PROGRAM PRG_Events
VAR
    aWarningEvents : ARRAY[0..4, 0..100] OF BOOL;
// 	sHeaterMinimum : STRING(32);
// 	sHeaterCurrent : STRING(32);
    fbEventsManager : FB_EventsManager;
    tonUpSupplyLost : TON;
    tonUsSupplyLost : TON;
    ton48VSupplyLost : TON;
    tonIndexPositionInvalid : TON;

    // Short-lived operator feedback for Heat Stake settings transactions.
    tpHeatStakeSettingsSaved : TP;
    tpHeatStakeSettingsRejected : TP;
    tpHeatStakeSettingsSaveFailed : TP;
END_VAR

GVL_MASTER.stStationEvents[0].aEvents[0].bFault := TRUE;
GVL_MASTER.stStationEvents[0].aEvents[0].bEventFlag :=
    (NOT GVL_MASTER.stInputs.bEmergencyStopChannel1 OR NOT GVL_MASTER.stInputs.bEmergencyStopChannel2)
    AND NOT GVL_MASTER.stInputs.stSafety.bSafetyOk;
GVL_MASTER.stStationEvents[0].aEvents[0].bEventText := 'E-stop activated';
GVL_MASTER.stStationEvents[0].aEvents[0].sSolution := 'Release E-stop and reset Safety';

GVL_MASTER.stStationEvents[0].aEvents[1].bFault := TRUE;
GVL_MASTER.stStationEvents[0].aEvents[1].bEventFlag :=
    (NOT GVL_MASTER.stInputs.bMainDoorChannel1 OR NOT GVL_MASTER.stInputs.bMainDoorChannel2)
    AND NOT GVL_MASTER.stInputs.stSafety.bSafetyOk;
GVL_MASTER.stStationEvents[0].aEvents[1].bEventText := 'Main door safety circuit open';
GVL_MASTER.stStationEvents[0].aEvents[1].sSolution := 'Close main door and reset Safety';


GVL_MASTER.stStationEvents[0].aEvents[2].bFault := TRUE;
GVL_MASTER.stStationEvents[0].aEvents[2].bEventFlag :=
    (NOT GVL_MASTER.stInputs.bLeftFlapChannel1 OR NOT GVL_MASTER.stInputs.bLeftFlapChannel2)
    AND NOT GVL_MASTER.stInputs.stSafety.bSafetyOk
    AND (GVL_MASTER.stStatus.eMachineState <> E_MachineState.PowerUp);
GVL_MASTER.stStationEvents[0].aEvents[2].bEventText := 'Right safety flap active';
GVL_MASTER.stStationEvents[0].aEvents[2].sSolution := 'Clear right flap and reset Safety';


GVL_MASTER.stStationEvents[0].aEvents[3].bFault := TRUE;
GVL_MASTER.stStationEvents[0].aEvents[3].bEventFlag :=
    (NOT GVL_MASTER.stInputs.bRightFlapChannel1 OR NOT GVL_MASTER.stInputs.bRightFlapChannel2)
    AND NOT GVL_MASTER.stInputs.stSafety.bSafetyOk
    AND (GVL_MASTER.stStatus.eMachineState <> E_MachineState.PowerUp);
GVL_MASTER.stStationEvents[0].aEvents[3].bEventText := 'Left safety flap active';
GVL_MASTER.stStationEvents[0].aEvents[3].sSolution := 'Clear left flap and reset Safety';


GVL_MASTER.stStationEvents[0].aEvents[4].bCycleStopRequest := TRUE;
GVL_MASTER.stStationEvents[0].aEvents[4].bEventFlag := GVL_MASTER.stCommand.bStop;
GVL_MASTER.stStationEvents[0].aEvents[4].bEventText := 'Cycle stop requested';
GVL_MASTER.stStationEvents[0].aEvents[4].sSolution := 'Wait for cycle to stop';

GVL_MASTER.stStationEvents[0].aEvents[5].bFault := TRUE;
GVL_MASTER.stStationEvents[0].aEvents[5].bEventFlag := GVL_MASTER.stStatus.bInitialisationTimeoutFault;
GVL_MASTER.stStationEvents[0].aEvents[5].bEventText := 'System initialisation timeout';
GVL_MASTER.stStationEvents[0].aEvents[5].sSolution := 'Check initialisation conditions';


GVL_MASTER.stStationEvents[0].aEvents[6].bFault := TRUE;
GVL_MASTER.stStationEvents[0].aEvents[6].bEventFlag := GVL_MASTER.stStatus.bStoppingTimeoutFault;
GVL_MASTER.stStationEvents[0].aEvents[6].bEventText := 'System stopping timeout';
GVL_MASTER.stStationEvents[0].aEvents[6].sSolution := 'Check index and machine safe state';


// Main-door supervision already causes immediate Fault; expose its actual cause.
GVL_MASTER.stStationEvents[0].aEvents[22].bFault := TRUE;
GVL_MASTER.stStationEvents[0].aEvents[22].bCycleStopRequest := FALSE;
GVL_MASTER.stStationEvents[0].aEvents[22].bEventFlag := GVL_MASTER.stStatus.stMainDoorLock.bFaulted;
GVL_MASTER.stStationEvents[0].aEvents[22].bEventText := CONCAT('Main door: ', GVL_MASTER.stStatus.stMainDoorLock.sMessage);
GVL_MASTER.stStationEvents[0].aEvents[22].sSolution := 'Check door/lock feedback and requested lock state; correct cause before Reset.';

tonUpSupplyLost(IN := NOT GVL_MASTER.stInputs.bUp24VPowerSupplyOk AND (GVL_MASTER.stStatus.eMachineState <> E_MachineState.PowerUp), PT := T#1S);

GVL_MASTER.stStationEvents[0].aEvents[7].bFault := TRUE;
GVL_MASTER.stStationEvents[0].aEvents[7].bEventFlag := tonUpSupplyLost.Q;
GVL_MASTER.stStationEvents[0].aEvents[7].bEventText := '24 V Up supply fault';
GVL_MASTER.stStationEvents[0].aEvents[7].sSolution := 'Check 24 V Up power supply';


tonUsSupplyLost(IN := NOT GVL_MASTER.stInputs.bUs24VPowerSupplyOk AND (GVL_MASTER.stStatus.eMachineState <> E_MachineState.PowerUp), PT := T#1S);

GVL_MASTER.stStationEvents[0].aEvents[8].bFault := TRUE;
GVL_MASTER.stStationEvents[0].aEvents[8].bEventFlag := tonUsSupplyLost.Q;
GVL_MASTER.stStationEvents[0].aEvents[8].bEventText := '24 V Us supply fault';
GVL_MASTER.stStationEvents[0].aEvents[8].sSolution := 'Check 24 V Us power supply';


ton48VSupplyLost(IN := NOT GVL_MASTER.stInputs.b48VPowerSupplyOk AND (GVL_MASTER.stStatus.eMachineState <> E_MachineState.PowerUp), PT := T#1S);

GVL_MASTER.stStationEvents[0].aEvents[9].bFault := TRUE;
GVL_MASTER.stStationEvents[0].aEvents[9].bEventFlag := ton48VSupplyLost.Q;
GVL_MASTER.stStationEvents[0].aEvents[9].bEventText := '48 V Up supply fault';
GVL_MASTER.stStationEvents[0].aEvents[9].sSolution := 'Check 48 V power supply';


tonIndexPositionInvalid(IN := GVL_MASTER.stInputs.bIndexReady AND GVL_MASTER.stInputs.bIndexLocked AND (GVL_MASTER.stInputs.eIndexPosition = E_TablePosition.Unknown), PT := T#500MS);

GVL_MASTER.stStationEvents[2].aEvents[0].bFault := TRUE;
GVL_MASTER.stStationEvents[2].aEvents[0].bEventFlag := tonIndexPositionInvalid.Q;
GVL_MASTER.stStationEvents[2].aEvents[0].bEventText := 'Index position sensors invalid';
GVL_MASTER.stStationEvents[2].aEvents[0].sSolution := 'Check index position sensors';



// -----------------------------------------------------------------------------
// PATCH PRESS STATION SUPPORT CYLINDERS
// Station group [3] is reserved here for process-station pneumatic faults.
// Each event is a machine fault and therefore participates in the existing
// bEventFault -> bSafetyDropRequest -> Immediate Fault chain.
// -----------------------------------------------------------------------------

// Patch Dispense support cylinder.
GVL_MASTER.stStationEvents[3].aEvents[0].bFault := TRUE;
GVL_MASTER.stStationEvents[3].aEvents[0].bEventFlag :=
    GVL_MASTER.stStatus.stPatchDispense.eSupportFault = E_SupportCylinderFault.ExtendTimeout;
GVL_MASTER.stStationEvents[3].aEvents[0].bEventText := 'Patch Dispense support cylinder UP feedback timeout';
GVL_MASTER.stStationEvents[3].aEvents[0].sSolution := 'Check UP sensor, air pressure, tubing, valve and cylinder mechanics';

GVL_MASTER.stStationEvents[3].aEvents[1].bFault := TRUE;
GVL_MASTER.stStationEvents[3].aEvents[1].bEventFlag :=
    GVL_MASTER.stStatus.stPatchDispense.eSupportFault = E_SupportCylinderFault.RetractTimeout;
GVL_MASTER.stStationEvents[3].aEvents[1].bEventText := 'Patch Dispense support cylinder DOWN feedback timeout';
GVL_MASTER.stStationEvents[3].aEvents[1].sSolution := 'Check DOWN sensor, air pressure, tubing, valve and cylinder mechanics';

GVL_MASTER.stStationEvents[3].aEvents[2].bFault := TRUE;
GVL_MASTER.stStationEvents[3].aEvents[2].bEventFlag :=
    GVL_MASTER.stStatus.stPatchDispense.eSupportFault = E_SupportCylinderFault.ContradictorySensors;
GVL_MASTER.stStationEvents[3].aEvents[2].bEventText := 'Patch Dispense support cylinder sensor conflict';
GVL_MASTER.stStationEvents[3].aEvents[2].sSolution := 'Check support-cylinder UP/DOWN sensors and mechanical adjustment';

// Generic process-station faults.
// Support-cylinder faults already have their own more specific alarms below,
// therefore these generic events are active only when no support fault exists.

GVL_MASTER.stStationEvents[3].aEvents[9].bFault := TRUE;
GVL_MASTER.stStationEvents[3].aEvents[9].bEventFlag :=
    GVL_MASTER.stStatus.stPatchDispense.bFault
    AND (GVL_MASTER.stStatus.stPatchDispense.eSupportFault = E_SupportCylinderFault.None);
GVL_MASTER.stStationEvents[3].aEvents[9].bEventText := GVL_MASTER.stStatus.stPatchDispense.sDiagnostic;
GVL_MASTER.stStationEvents[3].aEvents[9].sSolution :=
    'Check Patch Dispense station diagnostic, process equipment and simulation fault request';

GVL_MASTER.stStationEvents[3].aEvents[10].bFault := TRUE;
GVL_MASTER.stStationEvents[3].aEvents[10].bEventFlag :=
    GVL_MASTER.stStatus.stHeatStake.bFault
    AND (GVL_MASTER.stStatus.stHeatStake.eSupportFault = E_SupportCylinderFault.None);
GVL_MASTER.stStationEvents[3].aEvents[10].bEventText := 'Heat Stake station fault';
GVL_MASTER.stStationEvents[3].aEvents[10].sSolution :=
    'Check Heat Stake station diagnostic, process equipment and simulation fault request';

GVL_MASTER.stStationEvents[3].aEvents[11].bFault := TRUE;
GVL_MASTER.stStationEvents[3].aEvents[11].bEventFlag :=
    GVL_MASTER.stStatus.stVision.bFault;
GVL_MASTER.stStationEvents[3].aEvents[11].bEventText := 'Vision station fault';
GVL_MASTER.stStationEvents[3].aEvents[11].sSolution :=
    'Check Vision station diagnostic, process equipment and simulation fault request';

// =====================================================
// EVENT 12 - HEAT STAKE LOW TEMPERATURE WARNING
// =====================================================

// // Convert live temperature values to text.
// sHeaterMinimum := LREAL_TO_STRING(
//     GVL_MASTER.stStatus.stHeatStakeTemperature.rLowLimitC
// );
// 
// sHeaterCurrent := LREAL_TO_STRING(
//     GVL_MASTER.stStatus.stHeatStakeTemperature.rOverTempTemperatureC
// );
// 
// // Warning configuration.
// GVL_MASTER.stStationEvents[3].aEvents[12].bFault := FALSE;
// GVL_MASTER.stStationEvents[3].aEvents[12].bMessage := TRUE;
// GVL_MASTER.stStationEvents[3].aEvents[12].bPersistentMessage := TRUE;
// 
// // Active during AutoCycle and Dwell when temperature is low.
// GVL_MASTER.stStationEvents[3].aEvents[12].bEventFlag :=
//     (
//         (GVL_MASTER.stStatus.eMachineState = E_MachineState.AutoCycle)
//         OR (GVL_MASTER.stStatus.eMachineState = E_MachineState.Dwell)
//     )
//     AND NOT GVL_MASTER.stStatus.stHeatStakeTemperature.bIndexTemperatureReady;
// 
// // Dynamic warning message.
// GVL_MASTER.stStationEvents[3].aEvents[12].bEventText :=
//                 'Heater Temp below min - Min: ';
// GVL_MASTER.stStationEvents[3].aEvents[12].sSolution :=
//     CONCAT(
//         CONCAT(
//             CONCAT(
//                 'Low Limit Temp: ',
//                 sHeaterMinimum
//             ),
//             ' C | Current Temp: '
//         ),
//         sHeaterCurrent
//     );

GVL_MASTER.stStationEvents[3].aEvents[13].bFault :=FALSE;
GVL_MASTER.stStationEvents[3].aEvents[13].bEventFlag := 
    GVL_MASTER.stStatus.stHeatStakeTemperature.bLowTemperatureTimeout;
GVL_MASTER.stStationEvents[3].aEvents[13].bEventText :=
    'Heat Stake low temperature timeout';
GVL_MASTER.stStationEvents[3].aEvents[13].sSolution :=
    'Check heaters, SSRs, EL2502 outputs, thermocouples and temperature control';

GVL_MASTER.stStationEvents[3].aEvents[14].bFault := TRUE;
GVL_MASTER.stStationEvents[3].aEvents[14].bEventFlag :=
    GVL_MASTER.stStatus.stHeatStakeTemperature.bHighTemperature;
GVL_MASTER.stStationEvents[3].aEvents[14].bEventText :=
    'Heat Stake process temperature above high limit';
GVL_MASTER.stStationEvents[3].aEvents[14].sSolution :=
    'Heater power is disabled; wait for temperature to fall below the configured high limit before Reset';

GVL_MASTER.stStationEvents[3].aEvents[15].bFault := TRUE;
GVL_MASTER.stStationEvents[3].aEvents[15].bEventFlag :=
    GVL_MASTER.stStatus.stHeatStakeTemperature.bTemperatureDiscrepancy;
GVL_MASTER.stStationEvents[3].aEvents[15].bEventText :=
    'Heat Stake thermocouple temperature discrepancy';
GVL_MASTER.stStationEvents[3].aEvents[15].sSolution :=
    'Check both heater thermocouples, heater power and thermal contact';

GVL_MASTER.stStationEvents[3].aEvents[16].bFault := TRUE;
GVL_MASTER.stStationEvents[3].aEvents[16].bEventFlag :=
    GVL_MASTER.stStatus.stHeatStakeTemperature.bOverTemperature;
GVL_MASTER.stStationEvents[3].aEvents[16].bEventText :=
    'Heat Stake independent overtemperature active';
GVL_MASTER.stStationEvents[3].aEvents[16].sSolution :=
    'Heater power is disabled; temperature must fall below 90 C before Safety Reset is accepted';

GVL_MASTER.stStationEvents[3].aEvents[17].bFault := TRUE;
GVL_MASTER.stStationEvents[3].aEvents[17].bEventFlag :=
    GVL_MASTER.stStatus.stHeatStakeTemperature.bPid1Fault
    OR GVL_MASTER.stStatus.stHeatStakeTemperature.bPid2Fault;
GVL_MASTER.stStationEvents[3].aEvents[17].bEventText :=
    'Heat Stake temperature controller fault';
GVL_MASTER.stStationEvents[3].aEvents[17].sSolution :=
    'Check TF4100 Controller Toolbox parameters and PID diagnostics';

// -----------------------------------------------------------------------------
// HEAT STAKE SETTINGS APPLY / PERSISTENCE RESULT
// -----------------------------------------------------------------------------
//
// FB_EventsManager treats ordinary Messages as history-only.
// bPersistentMessage makes a Message visible in astActiveEvents[1..50] while
// bEventFlag is TRUE. Therefore these transaction results are converted into
// short TP windows: they are visible to the operator for a few seconds and are
// also written once into the event history.
//
// The source status bits may remain latched for diagnostics; the TP guarantees
// that the active DataGrid indication clears automatically.

// Generate short display windows on the rising edge of each transaction result.
tpHeatStakeSettingsSaveFailed(
    IN := GVL_HMI.stStatus.bHeatStakeSettingsSaveFailed,
    PT := T#5S
);

tpHeatStakeSettingsSaved(
    IN := GVL_HMI.stStatus.bHeatStakeSettingsSaveSuccessful,
    PT := T#3S
);

tpHeatStakeSettingsRejected(
    IN := GVL_HMI.stStatus.bHeatStakeSettingsApplyRejected,
    PT := T#5S
);

// Final persistence failure.
GVL_MASTER.stStationEvents[3].aEvents[18].bFault := FALSE;
GVL_MASTER.stStationEvents[3].aEvents[18].bMessage := TRUE;
GVL_MASTER.stStationEvents[3].aEvents[18].bPersistentMessage := TRUE;
GVL_MASTER.stStationEvents[3].aEvents[18].bEventFlag :=
    tpHeatStakeSettingsSaveFailed.Q;
GVL_MASTER.stStationEvents[3].aEvents[18].bEventText :=
    'Heat Stake settings save failed';
GVL_MASTER.stStationEvents[3].aEvents[18].sSolution :=
    'Check persistent-data access and Heat Stake settings write error ID';

// Successful save.
GVL_MASTER.stStationEvents[3].aEvents[19].bFault := FALSE;
GVL_MASTER.stStationEvents[3].aEvents[19].bMessage := TRUE;
GVL_MASTER.stStationEvents[3].aEvents[19].bPersistentMessage := TRUE;
GVL_MASTER.stStationEvents[3].aEvents[19].bEventFlag :=
    tpHeatStakeSettingsSaved.Q;
GVL_MASTER.stStationEvents[3].aEvents[19].bEventText :=
    'Heat Stake settings saved successfully';
GVL_MASTER.stStationEvents[3].aEvents[19].sSolution :=
    'No action required';

// Apply request rejected.
GVL_MASTER.stStationEvents[3].aEvents[20].bFault := FALSE;
GVL_MASTER.stStationEvents[3].aEvents[20].bMessage := TRUE;
GVL_MASTER.stStationEvents[3].aEvents[20].bPersistentMessage := TRUE;
GVL_MASTER.stStationEvents[3].aEvents[20].bEventFlag :=
    tpHeatStakeSettingsRejected.Q;
GVL_MASTER.stStationEvents[3].aEvents[20].bEventText :=
    GVL_HMI.stStatus.sHeatStakeSettingsApplyRejectReason;
GVL_MASTER.stStationEvents[3].aEvents[20].sSolution :=
    'Correct the condition reported in the message and apply the settings again';

// Heat Stake support cylinder.
// Heat Stake head cylinder position feedback alarms
GVL_MASTER.stStationEvents[3].aEvents[21].bFault := TRUE;
GVL_MASTER.stStationEvents[3].aEvents[21].bEventFlag := GVL_MASTER.stStatus.bHeatStakeHeadDownTimeoutFault;
GVL_MASTER.stStationEvents[3].aEvents[21].bEventText := 'Heat Stake head failed to reach DOWN position';
GVL_MASTER.stStationEvents[3].aEvents[21].sSolution := 'Check part presence, nest support UP position, DOWN sensor, pneumatic pressure, valve and cylinder mechanics';

GVL_MASTER.stStationEvents[3].aEvents[22].bFault := TRUE;
GVL_MASTER.stStationEvents[3].aEvents[22].bEventFlag := GVL_MASTER.stStatus.bHeatStakeHeadUpTimeoutFault;
GVL_MASTER.stStationEvents[3].aEvents[22].bEventText := 'Heat Stake head failed to reach UP position';
GVL_MASTER.stStationEvents[3].aEvents[22].sSolution := 'Check UP sensor, pneumatic pressure, valve, tubing and cylinder mechanics';

GVL_MASTER.stStationEvents[3].aEvents[23].bFault := TRUE;
GVL_MASTER.stStationEvents[3].aEvents[23].bEventFlag := GVL_MASTER.stStatus.bHeatStakeHeadSensorConflictFault;
GVL_MASTER.stStationEvents[3].aEvents[23].bEventText := 'Heat Stake head position sensor conflict';
GVL_MASTER.stStationEvents[3].aEvents[23].sSolution := 'Check Head UP/DOWN sensor wiring, magnetic sensor adjustment and mechanical position';

// =====================================================
// EVENT 24 - HEAT STAKE DWELL TIMEOUT
// =====================================================

GVL_MASTER.stStationEvents[3].aEvents[24].bFault := TRUE;
GVL_MASTER.stStationEvents[3].aEvents[24].bEventFlag :=GVL_MASTER.stStatus.bHeaterDwellTimeoutFault;
GVL_MASTER.stStationEvents[3].aEvents[24].bEventText :='Dwell timeout - temperature did not recover';
GVL_MASTER.stStationEvents[3].aEvents[24].sSolution :='Check heaters, thermocouples and temperature settings.';

// -----------------------------------------------------------------------------
// VISION CAMERA RUN STATUS - LIVE OPERATOR MESSAGE
// -----------------------------------------------------------------------------
// Run_Status FALSE cannot distinguish Setup from an unavailable camera.
// Keep this visible until RUN returns; Reset must not hide an active condition.

// Camera evaluation errors reject the product without a machine fault.
GVL_MASTER.stStationEvents[3].aEvents[26].bFault := FALSE;
GVL_MASTER.stStationEvents[3].aEvents[26].bCycleStopRequest := FALSE;
GVL_MASTER.stStationEvents[3].aEvents[26].bMessage := TRUE;
GVL_MASTER.stStationEvents[3].aEvents[26].bPersistentMessage := FALSE;
aWarningEvents[3, 26] := TRUE;
GVL_MASTER.stStationEvents[3].aEvents[26].bEventFlag :=
    (PRG_Main.fbMachine.fbVSCamera.aInspectionError0[1] <> 0)
    OR (PRG_Main.fbMachine.fbVSCamera.aInspectionError1[1] <> 0);
GVL_MASTER.stStationEvents[3].aEvents[26].bEventText := 'Vision image 1: inspection FAIL';
// Preserve error details while the warning awaits Reset, even after a new piece.
IF GVL_MASTER.stStationEvents[3].aEvents[26].bEventFlag THEN
    GVL_MASTER.stStationEvents[3].aEvents[26].sSolution := CONCAT('Camera Error0=', UDINT_TO_STRING(PRG_Main.fbMachine.fbVSCamera.aInspectionError0[1]));
    GVL_MASTER.stStationEvents[3].aEvents[26].sSolution := CONCAT(GVL_MASTER.stStationEvents[3].aEvents[26].sSolution, ' Error1=');
    GVL_MASTER.stStationEvents[3].aEvents[26].sSolution := CONCAT(GVL_MASTER.stStationEvents[3].aEvents[26].sSolution, UDINT_TO_STRING(PRG_Main.fbMachine.fbVSCamera.aInspectionError1[1]));
END_IF

GVL_MASTER.stStationEvents[3].aEvents[27].bFault := FALSE;
GVL_MASTER.stStationEvents[3].aEvents[27].bCycleStopRequest := FALSE;
GVL_MASTER.stStationEvents[3].aEvents[27].bMessage := TRUE;
GVL_MASTER.stStationEvents[3].aEvents[27].bPersistentMessage := FALSE;
aWarningEvents[3, 27] := TRUE;
GVL_MASTER.stStationEvents[3].aEvents[27].bEventFlag :=
    (PRG_Main.fbMachine.fbVSCamera.aInspectionError0[2] <> 0)
    OR (PRG_Main.fbMachine.fbVSCamera.aInspectionError1[2] <> 0);
GVL_MASTER.stStationEvents[3].aEvents[27].bEventText := 'Vision image 2: inspection FAIL';
// Preserve error details while the warning awaits Reset, even after a new piece.
IF GVL_MASTER.stStationEvents[3].aEvents[27].bEventFlag THEN
    GVL_MASTER.stStationEvents[3].aEvents[27].sSolution := CONCAT('Camera Error0=', UDINT_TO_STRING(PRG_Main.fbMachine.fbVSCamera.aInspectionError0[2]));
    GVL_MASTER.stStationEvents[3].aEvents[27].sSolution := CONCAT(GVL_MASTER.stStationEvents[3].aEvents[27].sSolution, ' Error1=');
    GVL_MASTER.stStationEvents[3].aEvents[27].sSolution := CONCAT(GVL_MASTER.stStationEvents[3].aEvents[27].sSolution, UDINT_TO_STRING(PRG_Main.fbMachine.fbVSCamera.aInspectionError1[2]));
END_IF

GVL_MASTER.stStationEvents[3].aEvents[28].bFault := FALSE;
GVL_MASTER.stStationEvents[3].aEvents[28].bCycleStopRequest := FALSE;
GVL_MASTER.stStationEvents[3].aEvents[28].bMessage := TRUE;
GVL_MASTER.stStationEvents[3].aEvents[28].bPersistentMessage := FALSE;
aWarningEvents[3, 28] := TRUE;
GVL_MASTER.stStationEvents[3].aEvents[28].bEventFlag :=
    (PRG_Main.fbMachine.fbVSCamera.aInspectionError0[3] <> 0)
    OR (PRG_Main.fbMachine.fbVSCamera.aInspectionError1[3] <> 0);
GVL_MASTER.stStationEvents[3].aEvents[28].bEventText := 'Vision image 3: inspection FAIL';
// Preserve error details while the warning awaits Reset, even after a new piece.
IF GVL_MASTER.stStationEvents[3].aEvents[28].bEventFlag THEN
    GVL_MASTER.stStationEvents[3].aEvents[28].sSolution := CONCAT('Camera Error0=', UDINT_TO_STRING(PRG_Main.fbMachine.fbVSCamera.aInspectionError0[3]));
    GVL_MASTER.stStationEvents[3].aEvents[28].sSolution := CONCAT(GVL_MASTER.stStationEvents[3].aEvents[28].sSolution, ' Error1=');
    GVL_MASTER.stStationEvents[3].aEvents[28].sSolution := CONCAT(GVL_MASTER.stStationEvents[3].aEvents[28].sSolution, UDINT_TO_STRING(PRG_Main.fbMachine.fbVSCamera.aInspectionError1[3]));
END_IF

GVL_MASTER.stStationEvents[3].aEvents[29].bFault := FALSE;
GVL_MASTER.stStationEvents[3].aEvents[29].bCycleStopRequest := FALSE;
GVL_MASTER.stStationEvents[3].aEvents[29].bMessage := TRUE;
GVL_MASTER.stStationEvents[3].aEvents[29].bPersistentMessage := FALSE;
aWarningEvents[3, 29] := TRUE;
GVL_MASTER.stStationEvents[3].aEvents[29].bEventFlag :=
    (PRG_Main.fbMachine.fbVSCamera.aInspectionError0[4] <> 0)
    OR (PRG_Main.fbMachine.fbVSCamera.aInspectionError1[4] <> 0);
GVL_MASTER.stStationEvents[3].aEvents[29].bEventText := 'Vision image 4: inspection FAIL';
// Preserve error details while the warning awaits Reset, even after a new piece.
IF GVL_MASTER.stStationEvents[3].aEvents[29].bEventFlag THEN
    GVL_MASTER.stStationEvents[3].aEvents[29].sSolution := CONCAT('Camera Error0=', UDINT_TO_STRING(PRG_Main.fbMachine.fbVSCamera.aInspectionError0[4]));
    GVL_MASTER.stStationEvents[3].aEvents[29].sSolution := CONCAT(GVL_MASTER.stStationEvents[3].aEvents[29].sSolution, ' Error1=');
    GVL_MASTER.stStationEvents[3].aEvents[29].sSolution := CONCAT(GVL_MASTER.stStationEvents[3].aEvents[29].sSolution, UDINT_TO_STRING(PRG_Main.fbMachine.fbVSCamera.aInspectionError1[4]));
END_IF

// Recovery failure is an equipment problem, not an accepted product verdict.
GVL_MASTER.stStationEvents[3].aEvents[30].bFault := TRUE;
GVL_MASTER.stStationEvents[3].aEvents[30].bEventFlag := PRG_Main.fbMachine.fbVSCamera.bRecoveryFailed;
GVL_MASTER.stStationEvents[3].aEvents[30].bEventText := 'Vision camera recovery failed after inspection error';
GVL_MASTER.stStationEvents[3].aEvents[30].sSolution := 'Check camera RUN, error codes and trigger readiness; restore camera and reset machine.';

GVL_MASTER.stStationEvents[3].aEvents[25].bFault := FALSE;
GVL_MASTER.stStationEvents[3].aEvents[25].bCycleStopRequest := FALSE;
GVL_MASTER.stStationEvents[3].aEvents[25].bMessage := TRUE;
GVL_MASTER.stStationEvents[3].aEvents[25].bPersistentMessage := TRUE;
GVL_MASTER.stStationEvents[3].aEvents[25].bEventFlag :=
    GVL_MASTER.stStatus.stVision.bCommissioned
    AND NOT GVL_EtherCAT.stVSKeyenceCamera.bRunStatus;
GVL_MASTER.stStationEvents[3].aEvents[25].bEventText :=
    'Camera not in RUN mode';
GVL_MASTER.stStationEvents[3].aEvents[25].sSolution :=
    'In Manual Mode/Vision, click "Open Interface" and select RUN.';



GVL_MASTER.stStationEvents[3].aEvents[3].bFault := TRUE;
GVL_MASTER.stStationEvents[3].aEvents[3].bEventFlag :=
    GVL_MASTER.stStatus.stHeatStake.eSupportFault = E_SupportCylinderFault.ExtendTimeout;
GVL_MASTER.stStationEvents[3].aEvents[3].bEventText := 'Heat Stake support cylinder UP feedback timeout';
GVL_MASTER.stStationEvents[3].aEvents[3].sSolution := 'Check UP sensor, air pressure, tubing, valve and cylinder mechanics';

GVL_MASTER.stStationEvents[3].aEvents[4].bFault := TRUE;
GVL_MASTER.stStationEvents[3].aEvents[4].bEventFlag :=
    GVL_MASTER.stStatus.stHeatStake.eSupportFault = E_SupportCylinderFault.RetractTimeout;
GVL_MASTER.stStationEvents[3].aEvents[4].bEventText := 'Heat Stake support cylinder DOWN feedback timeout';
GVL_MASTER.stStationEvents[3].aEvents[4].sSolution := 'Check DOWN sensor, air pressure, tubing, valve and cylinder mechanics';

GVL_MASTER.stStationEvents[3].aEvents[5].bFault := TRUE;
GVL_MASTER.stStationEvents[3].aEvents[5].bEventFlag :=
    GVL_MASTER.stStatus.stHeatStake.eSupportFault = E_SupportCylinderFault.ContradictorySensors;
GVL_MASTER.stStationEvents[3].aEvents[5].bEventText := 'Heat Stake support cylinder sensor conflict';
GVL_MASTER.stStationEvents[3].aEvents[5].sSolution := 'Check support-cylinder UP/DOWN sensors and mechanical adjustment';

// Vision support cylinder.
GVL_MASTER.stStationEvents[3].aEvents[6].bFault := TRUE;
GVL_MASTER.stStationEvents[3].aEvents[6].bEventFlag := FALSE; // Vision nest support removed; keep alarm ID reserved.
GVL_MASTER.stStationEvents[3].aEvents[6].bEventText := 'Vision support cylinder UP feedback timeout';
GVL_MASTER.stStationEvents[3].aEvents[6].sSolution := 'Check UP sensor, air pressure, tubing, valve and cylinder mechanics';

GVL_MASTER.stStationEvents[3].aEvents[7].bFault := TRUE;
GVL_MASTER.stStationEvents[3].aEvents[7].bEventFlag := FALSE; // Vision nest support removed; keep alarm ID reserved.
GVL_MASTER.stStationEvents[3].aEvents[7].bEventText := 'Vision support cylinder DOWN feedback timeout';
GVL_MASTER.stStationEvents[3].aEvents[7].sSolution := 'Check DOWN sensor, air pressure, tubing, valve and cylinder mechanics';

GVL_MASTER.stStationEvents[3].aEvents[8].bFault := TRUE;
GVL_MASTER.stStationEvents[3].aEvents[8].bEventFlag := FALSE; // Vision nest support removed; keep alarm ID reserved.
GVL_MASTER.stStationEvents[3].aEvents[8].bEventText := 'Vision support cylinder sensor conflict';
GVL_MASTER.stStationEvents[3].aEvents[8].sSolution := 'Check support-cylinder UP/DOWN sensors and mechanical adjustment';

// =========================================================
// EVENT 20 - HMI LOGOUT DURING OPERATION
// =========================================================

GVL_MASTER.stStationEvents[0].aEvents[20].bFault := TRUE;
GVL_MASTER.stStationEvents[0].aEvents[20].bEventFlag :=GVL_HMI.bHmiLogoutAutoCycle;
GVL_MASTER.stStationEvents[0].aEvents[20].bEventText :='HMI communication lost or logout during operation';
GVL_MASTER.stStationEvents[0].aEvents[20].sSolution :=
    'Check HMI connection and heartbeat; log in and reset the machine';

// =========================================================
// EVENT 21 - HMI LOGOUT / NO USER LOGGED IN
// =========================================================

GVL_MASTER.stStationEvents[0].aEvents[21].bCycleStopRequest := TRUE;
GVL_MASTER.stStationEvents[0].aEvents[21].bEventFlag :=GVL_HMI.bHmiLogoutStopped;
GVL_MASTER.stStationEvents[0].aEvents[21].bEventText :='HMI logout or no user logged in';
GVL_MASTER.stStationEvents[0].aEvents[21].sSolution :='Log in to continue operation';

// -----------------------------------------------------------------------------
// INDEX TABLE COMPONENT FAULTS
// These faults are latched inside FB_IndexTable4 until Reset.
// They are explicit bFault events so every Immediate Fault caused by the index
// is visible in the standard Active Events DataGrid.
// -----------------------------------------------------------------------------

GVL_MASTER.stStationEvents[0].aEvents[10].bFault := TRUE;
GVL_MASTER.stStationEvents[0].aEvents[10].bEventFlag :=
    GVL_MASTER.stStatus.stIndexStatus.eFault = E_IndexFault.InitialPositionInvalid;
GVL_MASTER.stStationEvents[0].aEvents[10].bEventText := 'Index initial position invalid';
GVL_MASTER.stStationEvents[0].aEvents[10].sSolution := 'Check index position sensors and table mechanical position';

GVL_MASTER.stStationEvents[0].aEvents[11].bFault := TRUE;
GVL_MASTER.stStationEvents[0].aEvents[11].bEventFlag :=
    GVL_MASTER.stStatus.stIndexStatus.eFault = E_IndexFault.SupportRetractTimeout;
GVL_MASTER.stStationEvents[0].aEvents[11].bEventText := 'Index support retract timeout';
GVL_MASTER.stStationEvents[0].aEvents[11].sSolution := 'Check support feedback and pneumatic movement';

GVL_MASTER.stStationEvents[0].aEvents[12].bFault := TRUE;
GVL_MASTER.stStationEvents[0].aEvents[12].bEventFlag :=
    GVL_MASTER.stStatus.stIndexStatus.eFault = E_IndexFault.RotationTimeout;
GVL_MASTER.stStationEvents[0].aEvents[12].bEventText := 'Index rotation timeout';
GVL_MASTER.stStationEvents[0].aEvents[12].sSolution := 'Check index pneumatic supply, valve outputs and table movement';

GVL_MASTER.stStationEvents[0].aEvents[13].bFault := TRUE;
GVL_MASTER.stStationEvents[0].aEvents[13].bEventFlag :=
    GVL_MASTER.stStatus.stIndexStatus.eFault = E_IndexFault.StopAndLockTimeout;
GVL_MASTER.stStationEvents[0].aEvents[13].bEventText := 'Index stop / lock timeout';
GVL_MASTER.stStationEvents[0].aEvents[13].sSolution := 'Check Index Ready, Locked and Completed feedbacks';

GVL_MASTER.stStationEvents[0].aEvents[14].bFault := TRUE;
GVL_MASTER.stStationEvents[0].aEvents[14].bEventFlag :=
    GVL_MASTER.stStatus.stIndexStatus.eFault = E_IndexFault.PositionInvalid;
GVL_MASTER.stStationEvents[0].aEvents[14].bEventText := 'Index position invalid after movement';
GVL_MASTER.stStationEvents[0].aEvents[14].sSolution := 'Check index position sensors and final table position';

GVL_MASTER.stStationEvents[0].aEvents[15].bFault := TRUE;
GVL_MASTER.stStationEvents[0].aEvents[15].bEventFlag :=
    GVL_MASTER.stStatus.stIndexStatus.eFault = E_IndexFault.SupportExtendTimeout;
GVL_MASTER.stStationEvents[0].aEvents[15].bEventText := 'Index support extend timeout';
GVL_MASTER.stStationEvents[0].aEvents[15].sSolution := 'Check support feedback and pneumatic movement';

GVL_MASTER.stStationEvents[0].aEvents[16].bFault := TRUE;
GVL_MASTER.stStationEvents[0].aEvents[16].bEventFlag :=
    GVL_MASTER.stStatus.stIndexStatus.eFault = E_IndexFault.TwoHandReleasedDuringMovement;
GVL_MASTER.stStationEvents[0].aEvents[16].bEventText := 'Two-hand control released during index movement';
GVL_MASTER.stStationEvents[0].aEvents[16].sSolution := 'Hold both touch buttons until index movement is complete';

GVL_MASTER.stStationEvents[0].aEvents[17].bFault := TRUE;
GVL_MASTER.stStationEvents[0].aEvents[17].bEventFlag :=
    GVL_MASTER.stStatus.stIndexStatus.eFault = E_IndexFault.WrongPositionTimeout;
GVL_MASTER.stStationEvents[0].aEvents[17].bEventText := 'Index wrong-position recovery timeout';
GVL_MASTER.stStationEvents[0].aEvents[17].sSolution := 'Check table position sensors and index mechanical alignment';

GVL_MASTER.stStationEvents[0].aEvents[18].bFault := TRUE;
GVL_MASTER.stStationEvents[0].aEvents[18].bEventFlag :=
    GVL_MASTER.stStatus.stIndexStatus.eFault = E_IndexFault.SafetyLostDuringMovement;
GVL_MASTER.stStationEvents[0].aEvents[18].bEventText := 'Index motion safety lost during movement';
GVL_MASTER.stStationEvents[0].aEvents[18].sSolution := 'Check TwinSAFE motion permissive and safety devices';

GVL_MASTER.stStationEvents[0].aEvents[19].bFault := TRUE;
GVL_MASTER.stStationEvents[0].aEvents[19].bEventFlag :=
    GVL_MASTER.stStatus.stIndexStatus.eFault = E_IndexFault.MovementPermissiveLost;
GVL_MASTER.stStationEvents[0].aEvents[19].bEventText := 'Index movement permissive lost during movement';
GVL_MASTER.stStationEvents[0].aEvents[19].sSolution := 'Check support cylinders and index movement permissives';

// -----------------------------------------------------------------------------
// AUTOMATIC PROCESS CYCLE
// -----------------------------------------------------------------------------

GVL_MASTER.stStationEvents[1].aEvents[1].bFault := TRUE;
GVL_MASTER.stStationEvents[1].aEvents[1].bEventFlag :=
    GVL_MASTER.stStatus.bProcessCycleTimeoutFault;
GVL_MASTER.stStationEvents[1].aEvents[1].bEventText :=
    'Automatic process cycle timeout';
GVL_MASTER.stStationEvents[1].aEvents[1].sSolution :=
    'Check ProcessCycle state, index permissives and required station completion';

GVL_MASTER.stStationEvents[1].aEvents[0].bMessage := TRUE;
GVL_MASTER.stStationEvents[1].aEvents[0].bPersistentMessage := TRUE;
GVL_MASTER.stStationEvents[1].aEvents[0].bEventFlag := NOT GVL_MASTER.stStatus.bAllStationsCommissioned;
GVL_MASTER.stStationEvents[1].aEvents[0].bEventText := GVL_MASTER.stStatus.sAutoCycleBlockReason;
GVL_MASTER.stStationEvents[1].aEvents[0].sSolution := 'Commission Patch Dispense, Heat Stake and Vision stations';



// Patch feeding NC/PLCopen diagnostics, one event per motor.
GVL_MASTER.stStationEvents[3].aEvents[31].bFault := TRUE;
GVL_MASTER.stStationEvents[3].aEvents[31].bEventFlag :=
    GVL_Motion.AxisDriveMotor.bError AND NOT GVL_Motion.stPatchFeedStatus.bResetPending;
GVL_MASTER.stStationEvents[3].aEvents[31].bEventText := CONCAT('M1 Drive Motor: axis error ', UDINT_TO_STRING(GVL_Motion.AxisDriveMotor.udiErrorId));
GVL_MASTER.stStationEvents[3].aEvents[31].sSolution := 'Check NC and drive diagnostics; correct cause before operator Reset.';

GVL_MASTER.stStationEvents[3].aEvents[32].bFault := TRUE;
GVL_MASTER.stStationEvents[3].aEvents[32].bEventFlag :=
    GVL_Motion.AxisPatchFeedRollMotor.bError AND NOT GVL_Motion.stPatchFeedStatus.bResetPending;
GVL_MASTER.stStationEvents[3].aEvents[32].bEventText := CONCAT('M2 Patch Feed Roll: axis error ', UDINT_TO_STRING(GVL_Motion.AxisPatchFeedRollMotor.udiErrorId));
GVL_MASTER.stStationEvents[3].aEvents[32].sSolution := 'Check NC and drive diagnostics; correct cause before operator Reset.';

GVL_MASTER.stStationEvents[3].aEvents[33].bFault := TRUE;
GVL_MASTER.stStationEvents[3].aEvents[33].bEventFlag :=
    GVL_Motion.AxisWasteRollMotor.bError AND NOT GVL_Motion.stPatchFeedStatus.bResetPending;
GVL_MASTER.stStationEvents[3].aEvents[33].bEventText := CONCAT('M3 Waste Roll: axis error ', UDINT_TO_STRING(GVL_Motion.AxisWasteRollMotor.udiErrorId));
GVL_MASTER.stStationEvents[3].aEvents[33].sSolution := 'Check NC and drive diagnostics; correct cause before operator Reset.';

GVL_MASTER.stStationEvents[3].aEvents[34].bFault := TRUE;
GVL_MASTER.stStationEvents[3].aEvents[34].bEventFlag :=
    GVL_Motion.stPatchFeedStatus.bFault
    AND NOT GVL_Motion.AxisDriveMotor.bError
    AND NOT GVL_Motion.AxisPatchFeedRollMotor.bError
    AND NOT GVL_Motion.AxisWasteRollMotor.bError;
GVL_MASTER.stStationEvents[3].aEvents[34].bEventText := GVL_Motion.stPatchFeedStatus.sDiagnostic;
GVL_MASTER.stStationEvents[3].aEvents[34].sSolution := 'Check rocker sensors and motion timeout; do not repeatedly retry a jammed web.';

// Explicit commissioning indication; no fault is suppressed by this message.
GVL_MASTER.stStationEvents[3].aEvents[35].bMessage := TRUE;
GVL_MASTER.stStationEvents[3].aEvents[35].bPersistentMessage := TRUE;
GVL_MASTER.stStationEvents[3].aEvents[35].bEventFlag :=
    GVL_MASTER.stStatus.stPatchDispense.bCommissioned
    AND NOT GVL_Motion.stPatchFeedSettings.bUsePatchVerticalFeedback;
GVL_MASTER.stStationEvents[3].aEvents[35].bEventText := 'Patch vertical: TEMP timed mode';
GVL_MASTER.stStationEvents[3].aEvents[35].sSolution :=
    'No position feedback. Wire Input9/Input10, validate and restore feedback mode.';

// Missing load components are start-only warnings, never machine faults or cycle stops.
aWarningEvents[1, 2] := TRUE;
GVL_MASTER.stStationEvents[1].aEvents[2].bMessage := TRUE;
GVL_MASTER.stStationEvents[1].aEvents[2].bEventFlag :=
    GVL_MASTER.stStatus.stOperatorStation.bMissingPbupAlert;
GVL_MASTER.stStationEvents[1].aEvents[2].bEventText := 'Operator nest: PBUP missing';
GVL_MASTER.stStationEvents[1].aEvents[2].sSolution :=
    'Load the PBUP or remove the product. Release both hands before trying again.';
IF NOT GVL_MASTER.stStationEvents[1].aEvents[2].bEventFlag THEN
    GVL_MASTER.stStationEvents[1].aEvents[2].bActive := FALSE;
END_IF
aWarningEvents[1, 3] := TRUE;
GVL_MASTER.stStationEvents[1].aEvents[3].bMessage := TRUE;
GVL_MASTER.stStationEvents[1].aEvents[3].bEventFlag :=
    GVL_MASTER.stStatus.stOperatorStation.bMissingProductAlert;
GVL_MASTER.stStationEvents[1].aEvents[3].bEventText := 'Operator nest: product missing';
GVL_MASTER.stStationEvents[1].aEvents[3].sSolution :=
    'Load the product or remove the PBUP. Release both hands before trying again.';
IF NOT GVL_MASTER.stStationEvents[1].aEvents[3].bEventFlag THEN
    GVL_MASTER.stStationEvents[1].aEvents[3].bActive := FALSE;
END_IF

// Per-physical-nest live warnings; never request Fault or cycle stop.
aWarningEvents[3, 36] := TRUE;
GVL_MASTER.stStationEvents[3].aEvents[36].bFault := FALSE;
GVL_MASTER.stStationEvents[3].aEvents[36].bCycleStopRequest := FALSE;
GVL_MASTER.stStationEvents[3].aEvents[36].bMessage := TRUE;
GVL_MASTER.stStationEvents[3].aEvents[36].bPersistentMessage := TRUE;
GVL_MASTER.stStationEvents[3].aEvents[36].bEventFlag :=
    GVL_MASTER.stStatus.aNest[1].stHeatStakeResult.bValid
    AND (GVL_MASTER.stStatus.aNest[1].stHeatStakeResult.udiAlertCode = GVL_MASTER.udiHeatStakePatchMissingAlertCode);
GVL_MASTER.stStationEvents[3].aEvents[36].bEventText := 'Nest 1: patch not detected at Heat Stake';
GVL_MASTER.stStationEvents[3].aEvents[36].sSolution := 'Heat Stake FAIL / Vision NOT TESTED. Reject this product at Operator; warning clears on confirmed reject.';

aWarningEvents[3, 37] := TRUE;
GVL_MASTER.stStationEvents[3].aEvents[37].bFault := FALSE;
GVL_MASTER.stStationEvents[3].aEvents[37].bCycleStopRequest := FALSE;
GVL_MASTER.stStationEvents[3].aEvents[37].bMessage := TRUE;
GVL_MASTER.stStationEvents[3].aEvents[37].bPersistentMessage := TRUE;
GVL_MASTER.stStationEvents[3].aEvents[37].bEventFlag :=
    GVL_MASTER.stStatus.aNest[2].stHeatStakeResult.bValid
    AND (GVL_MASTER.stStatus.aNest[2].stHeatStakeResult.udiAlertCode = GVL_MASTER.udiHeatStakePatchMissingAlertCode);
GVL_MASTER.stStationEvents[3].aEvents[37].bEventText := 'Nest 2: patch not detected at Heat Stake';
GVL_MASTER.stStationEvents[3].aEvents[37].sSolution := 'Heat Stake FAIL / Vision NOT TESTED. Reject this product at Operator; warning clears on confirmed reject.';

aWarningEvents[3, 38] := TRUE;
GVL_MASTER.stStationEvents[3].aEvents[38].bFault := FALSE;
GVL_MASTER.stStationEvents[3].aEvents[38].bCycleStopRequest := FALSE;
GVL_MASTER.stStationEvents[3].aEvents[38].bMessage := TRUE;
GVL_MASTER.stStationEvents[3].aEvents[38].bPersistentMessage := TRUE;
GVL_MASTER.stStationEvents[3].aEvents[38].bEventFlag :=
    GVL_MASTER.stStatus.aNest[3].stHeatStakeResult.bValid
    AND (GVL_MASTER.stStatus.aNest[3].stHeatStakeResult.udiAlertCode = GVL_MASTER.udiHeatStakePatchMissingAlertCode);
GVL_MASTER.stStationEvents[3].aEvents[38].bEventText := 'Nest 3: patch not detected at Heat Stake';
GVL_MASTER.stStationEvents[3].aEvents[38].sSolution := 'Heat Stake FAIL / Vision NOT TESTED. Reject this product at Operator; warning clears on confirmed reject.';

aWarningEvents[3, 39] := TRUE;
GVL_MASTER.stStationEvents[3].aEvents[39].bFault := FALSE;
GVL_MASTER.stStationEvents[3].aEvents[39].bCycleStopRequest := FALSE;
GVL_MASTER.stStationEvents[3].aEvents[39].bMessage := TRUE;
GVL_MASTER.stStationEvents[3].aEvents[39].bPersistentMessage := TRUE;
GVL_MASTER.stStationEvents[3].aEvents[39].bEventFlag :=
    GVL_MASTER.stStatus.aNest[4].stHeatStakeResult.bValid
    AND (GVL_MASTER.stStatus.aNest[4].stHeatStakeResult.udiAlertCode = GVL_MASTER.udiHeatStakePatchMissingAlertCode);
GVL_MASTER.stStationEvents[3].aEvents[39].bEventText := 'Nest 4: patch not detected at Heat Stake';
GVL_MASTER.stStationEvents[3].aEvents[39].sSolution := 'Heat Stake FAIL / Vision NOT TESTED. Reject this product at Operator; warning clears on confirmed reject.';

// Live camera startup warning: Reset cannot hide an error still active in the camera.
aWarningEvents[3, 40] := TRUE;
GVL_MASTER.stStationEvents[3].aEvents[40].bFault := FALSE;
GVL_MASTER.stStationEvents[3].aEvents[40].bCycleStopRequest := FALSE;
GVL_MASTER.stStationEvents[3].aEvents[40].bMessage := TRUE;
GVL_MASTER.stStationEvents[3].aEvents[40].bPersistentMessage := TRUE;
GVL_MASTER.stStationEvents[3].aEvents[40].bEventFlag :=
    PRG_Main.fbMachine.bVisionCameraStartBlocked;
GVL_MASTER.stStationEvents[3].aEvents[40].bEventText :=
    'Vision camera requires recovery - new capture blocked';
GVL_MASTER.stStationEvents[3].aEvents[40].sSolution :=
    CONCAT('Camera Error0=', UDINT_TO_STRING(GVL_EtherCAT.udiVisionError0Code));
GVL_MASTER.stStationEvents[3].aEvents[40].sSolution :=
    CONCAT(GVL_MASTER.stStationEvents[3].aEvents[40].sSolution, ' Error1=');
GVL_MASTER.stStationEvents[3].aEvents[40].sSolution :=
    CONCAT(GVL_MASTER.stStationEvents[3].aEvents[40].sSolution, UDINT_TO_STRING(GVL_EtherCAT.udiVisionError1Code));
GVL_MASTER.stStationEvents[3].aEvents[40].sSolution :=
    CONCAT(GVL_MASTER.stStationEvents[3].aEvents[40].sSolution, '. Manual: use Camera Reset, verify RUN and retry. AutoCycle keeps its existing stop/fault recovery; mechanical faults require machine recovery.');

// Live warnings after an attempted manual index; clear with their conditions.
aWarningEvents[3, 41] := TRUE;
GVL_MASTER.stStationEvents[3].aEvents[41].bFault := FALSE;
GVL_MASTER.stStationEvents[3].aEvents[41].bCycleStopRequest := FALSE;
GVL_MASTER.stStationEvents[3].aEvents[41].bMessage := TRUE;
GVL_MASTER.stStationEvents[3].aEvents[41].bPersistentMessage := TRUE;
GVL_MASTER.stStationEvents[3].aEvents[41].bEventFlag := GVL_MASTER.bManualIndexBlockVision;
GVL_MASTER.stStationEvents[3].aEvents[41].bEventText := GVL_MASTER.sManualIndexVisionReason;
GVL_MASTER.stStationEvents[3].aEvents[41].sSolution := 'Return Vision HOME; if holding a part, prepare Image 4, then Release Position. Release two-hand and actuate again.';

aWarningEvents[3, 42] := TRUE;
GVL_MASTER.stStationEvents[3].aEvents[42].bFault := FALSE;
GVL_MASTER.stStationEvents[3].aEvents[42].bCycleStopRequest := FALSE;
GVL_MASTER.stStationEvents[3].aEvents[42].bMessage := TRUE;
GVL_MASTER.stStationEvents[3].aEvents[42].bPersistentMessage := TRUE;
GVL_MASTER.stStationEvents[3].aEvents[42].bEventFlag := GVL_MASTER.bManualIndexBlockHeat;
GVL_MASTER.stStationEvents[3].aEvents[42].bEventText := 'Index blocked: Heat Stake not HOME';
GVL_MASTER.stStationEvents[3].aEvents[42].sSolution := 'Return Heat Stake head UP/locked and nest support DOWN. Release two-hand and actuate again.';

aWarningEvents[3, 43] := TRUE;
GVL_MASTER.stStationEvents[3].aEvents[43].bFault := FALSE;
GVL_MASTER.stStationEvents[3].aEvents[43].bCycleStopRequest := FALSE;
GVL_MASTER.stStationEvents[3].aEvents[43].bMessage := TRUE;
GVL_MASTER.stStationEvents[3].aEvents[43].bPersistentMessage := TRUE;
GVL_MASTER.stStationEvents[3].aEvents[43].bEventFlag := GVL_MASTER.bManualIndexBlockPatch;
GVL_MASTER.stStationEvents[3].aEvents[43].bEventText := 'Index blocked: Patch tooling/feed not ready';
GVL_MASTER.stStationEvents[3].aEvents[43].sSolution := 'Return Patch transfer vertical UP and finish feeding/manual strokes. Release two-hand and actuate again.';

aWarningEvents[3, 44] := TRUE;
GVL_MASTER.stStationEvents[3].aEvents[44].bFault := FALSE;
GVL_MASTER.stStationEvents[3].aEvents[44].bCycleStopRequest := FALSE;
GVL_MASTER.stStationEvents[3].aEvents[44].bMessage := TRUE;
GVL_MASTER.stStationEvents[3].aEvents[44].bPersistentMessage := TRUE;
GVL_MASTER.stStationEvents[3].aEvents[44].bEventFlag := GVL_MASTER.bManualIndexBlockOther;
GVL_MASTER.stStationEvents[3].aEvents[44].bEventText := GVL_MASTER.sManualIndexOtherReason;
GVL_MASTER.stStationEvents[3].aEvents[44].sSolution := 'Correct the displayed index condition. No start is queued; release two-hand and actuate again.';

aWarningEvents[3, 45] := TRUE;
GVL_MASTER.stStationEvents[3].aEvents[45].bFault := FALSE;
GVL_MASTER.stStationEvents[3].aEvents[45].bCycleStopRequest := FALSE;
GVL_MASTER.stStationEvents[3].aEvents[45].bMessage := TRUE;
GVL_MASTER.stStationEvents[3].aEvents[45].bPersistentMessage := TRUE;
GVL_MASTER.stStationEvents[3].aEvents[45].bEventFlag := GVL_MASTER.bManualCameraRecoveryFailed;
GVL_MASTER.stStationEvents[3].aEvents[45].bEventText := 'Manual camera recovery failed - no capture sent';
GVL_MASTER.stStationEvents[3].aEvents[45].sSolution := 'Check camera error/RUN/handshake. Camera Reset recovers only; Camera Trigger may recover then capture. Machine Reset is not used.';

aWarningEvents[3, 46] := TRUE;
GVL_MASTER.stStationEvents[3].aEvents[46].bFault := FALSE;
GVL_MASTER.stStationEvents[3].aEvents[46].bCycleStopRequest := FALSE;
GVL_MASTER.stStationEvents[3].aEvents[46].bMessage := TRUE;
GVL_MASTER.stStationEvents[3].aEvents[46].bPersistentMessage := TRUE;
GVL_MASTER.stStationEvents[3].aEvents[46].bEventFlag := GVL_MASTER.bVisionManualCameraWarning;
GVL_MASTER.stStationEvents[3].aEvents[46].bEventText := 'Manual capture incomplete - camera recovery required';
GVL_MASTER.stStationEvents[3].aEvents[46].sSolution := 'Image 2: wait for return to 0 deg, then Camera Reset and retry Trigger. Tooling faults still require machine recovery.';

aWarningEvents[3, 47] := TRUE;
GVL_MASTER.stStationEvents[3].aEvents[47].bFault := FALSE;
GVL_MASTER.stStationEvents[3].aEvents[47].bCycleStopRequest := FALSE;
GVL_MASTER.stStationEvents[3].aEvents[47].bMessage := TRUE;
GVL_MASTER.stStationEvents[3].aEvents[47].bPersistentMessage := TRUE;
GVL_MASTER.stStationEvents[3].aEvents[47].bEventFlag := GVL_MASTER.bVisionManualGridWarning;
GVL_MASTER.stStationEvents[3].aEvents[47].bEventText := GVL_HMI.sCameraManualMessage;
GVL_MASTER.stStationEvents[3].aEvents[47].sSolution := CONCAT(GVL_HMI.sVisionPbupStatus, CONCAT(' | ', GVL_HMI.sVisionPbupSaveStatus));

aWarningEvents[3, 48] := FALSE;
GVL_MASTER.stStationEvents[3].aEvents[48].bFault := FALSE;
GVL_MASTER.stStationEvents[3].aEvents[48].bCycleStopRequest := FALSE;
GVL_MASTER.stStationEvents[3].aEvents[48].bMessage := TRUE;
GVL_MASTER.stStationEvents[3].aEvents[48].bPersistentMessage := TRUE;
GVL_MASTER.stStationEvents[3].aEvents[48].bEventFlag := GVL_MASTER.bVisionManualGridActive AND NOT GVL_MASTER.bVisionManualGridWarning
    AND NOT GVL_MASTER.bVisionManualCameraWarning AND NOT GVL_MASTER.bManualCameraRecoveryFailed
    AND (NOT PRG_Main.fbMachine.bVisionCameraStartBlocked OR PRG_Main.fbMachine.bManualCameraRecoveryActive);
GVL_MASTER.stStationEvents[3].aEvents[48].bEventText := GVL_HMI.sCameraManualMessage;
GVL_MASTER.stStationEvents[3].aEvents[48].sSolution := CONCAT(GVL_HMI.sVisionPbupStatus, CONCAT(' | ', GVL_HMI.sVisionPbupSaveStatus));

aWarningEvents[3, 49] := TRUE;
GVL_MASTER.stStationEvents[3].aEvents[49].bFault := FALSE;
GVL_MASTER.stStationEvents[3].aEvents[49].bCycleStopRequest := FALSE;
GVL_MASTER.stStationEvents[3].aEvents[49].bMessage := TRUE;
GVL_MASTER.stStationEvents[3].aEvents[49].bPersistentMessage := TRUE;
GVL_MASTER.stStationEvents[3].aEvents[49].bEventFlag := GVL_HMI.bVisionPbupSaveError;
GVL_MASTER.stStationEvents[3].aEvents[49].bEventText := 'PBUP state not saved';
GVL_MASTER.stStationEvents[3].aEvents[49].sSolution := GVL_HMI.sVisionPbupSaveStatus;

fbEventsManager(	aWarningEvents := aWarningEvents,
                    bPulse := TRUE,
					bDataWritedInCSV := FALSE, 
					nArraySize := 4, 
					bMachineMessage := GVL_MASTER.stStatus.sMachineMessage, 
					eMachineState := GVL_MASTER.stStatus.eMachineState, 
					stStationEvents := GVL_MASTER.stStationEvents, 
					stEventsAssigment := GVL_MASTER.stEventsAssigment, 
					bResetFaults := GVL_MASTER.stCommand.bReset, 
					bMachineFault => GVL_MASTER.bMachineFault, 
					bCycleStopRequest => GVL_MASTER.bCycleStopRequest, 
					sSystemDate => GVL_MASTER.sSystemDate,
					sSystemTime => GVL_MASTER.sSystemTime,
					astActiveEvents => GVL_MASTER.astActiveEvents, 
					astEventsHistory => GVL_Persistent.astEventsHistory
				);

// Expose Event Manager clock for HMI diagnostics/header use.
GVL_HMI.sSystemDate := GVL_MASTER.sSystemDate;
GVL_HMI.sSystemTime := GVL_MASTER.sSystemTime;

GVL_HMI.astActiveEvents := GVL_MASTER.astActiveEvents;
GVL_HMI.astEventsHistory := GVL_Persistent.astEventsHistory;
GVL_HMI.stEventsAssigment := GVL_MASTER.stEventsAssigment;

END_PROGRAM

(* stored: Version 1.1.0.1, ProductVersion 3.1.4026.18
   POU PRG_Events: Id {d91f2867-40c6-48eb-9107-f41ea1d35528}, SpecialFunc None *)
